TEXTLIST TL_MarkMode
  0 = 'AutoDefault'
  1 = 'None / Sim'
  2 = 'OneDefault'
  3 = 'OneTriangle'
   = ''
END_TEXTLIST

(* stored: Version 1.1.0.1, ProductVersion 3.1.4024.11
   TextList TL_MarkMode: Id {733d61ea-fd32-4d6a-b687-cbec33a52231} *)
